FUNCTION_BLOCK FB_IODEV_CH_DIG_OUT EXTENDS FB_IODEV_CH_DIGITAL
VAR_INPUT
END_VAR
VAR_OUTPUT
END_VAR
VAR
	// Physical active output signal.
	// Read-Only access via OPC UA.
	{attribute 'OPC.UA.DA' := '1'}
	{attribute 'OPC.UA.DA.Access' := '1'}
	q_bValue	AT %Q*:	BOOL;

	// Set values 
	// Configured for R/W OPC UA Data Access !!!
	{attribute 'OPC.UA.DA' := '1'}
	{attribute 'OPC.UA.DA.Access' := '3'}
	bValue:		BOOL;
	{attribute 'OPC.UA.DA' := '1'}
	{attribute 'OPC.UA.DA.Access' := '3'}
	sValueUser:	STRING(16);
	
	// Configuration parameters
	// Configured for R/W OPC UA Data Access !!!
	{attribute 'OPC.UA.DA' := '1'}
	{attribute 'OPC.UA.DA.Access' := '3'}
	nConversion:	E_IODEV_CONVERSION	:= CONVERSION_IODEV_NONE;
END_VAR

METHOD M_Compute
VAR_INPUT
END_VAR
// Check if the digital output should be calculated from User labels.
// If yes, convert user label to digital output value.
// Otherwise, just take the value from bValue and set the labels.
IF nConversion = CONVERSION_IODEV_DIGITAL THEN
	IF sValueUser = sLabel_0 THEN
		bValue	:= FALSE;
	ELSIF sValueUser = sLabel_1 THEN
		bValue	:= TRUE;
	END_IF
ELSE
	IF bValue THEN
		sValueUser	:= sLabel_1;
	ELSE
		sValueUser	:= sLabel_0;
	END_IF
END_IF

// Set output
q_bValue	:= bValue;
END_METHOD

METHOD M_Configure
VAR_INPUT
	in_nConversion:	INT			:= CONVERSION_IODEV_NONE;	// CONVERSION_IODEV_NONE or CONVERSION_IODEV_DIGITAL
	in_sLabel_0:	STRING(16)	:= '0';
	in_sLabel_1:	STRING(16)	:= '1';
END_VAR
// Set conversion type
nConversion	:= in_nConversion;

// Set labels
sLabel_0	:= in_sLabel_0;
sLabel_1	:= in_sLabel_1;

// Set output to zero
q_bValue	:= FALSE;
bValue		:= FALSE;
sValueUser	:= sLabel_0;
END_METHOD

METHOD M_Reset
VAR_INPUT
END_VAR
nConversion	:= CONVERSION_IODEV_NONE;
sLabel_0	:= '0';
sLabel_1	:= '1';

// Set output to zero
q_bValue	:= FALSE;
bValue		:= FALSE;
sValueUser	:= sLabel_0;
END_METHOD

END_FUNCTION_BLOCK

(* stored: Version 1.1.0.1, ProductVersion 3.1.4024.12
   POU FB_IODEV_CH_DIG_OUT: Id {2a8b35bb-758b-415b-8c12-01ef230835b1}, SpecialFunc None
   Method M_Compute: Id {8c77a573-dcab-4db3-b31d-c9208b3657b4}
   Method M_Configure: Id {fb6811ef-9e81-4d6a-99d3-56936a031f0e}
   Method M_Reset: Id {58226345-a012-4b10-b36c-b34f78a00873} *)
